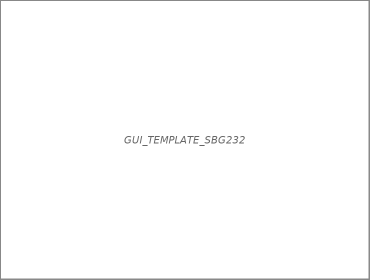
VISUALIZATION GUI_SBG232  // 370x280
    Frame (0,0 370x280)
        shows GUI_TEMPLATE_SBG232(m_Instance := MAIN.sbg232)
END_VISUALIZATION

(* stored: Version 1.1.0.1, ProductVersion 3.1.4024.12
   Visu GUI_SBG232: Id {578cf19f-63ce-4fbd-a11e-24fda4dbee82} *)
